FUNCTION_BLOCK Jack_Sledge_Place (* Composite Function Block Type *)
  (* Standard: 61499-2 *)
  (* Version 0.0, 4/24/2020, prana, nxtControl GmbH, template *)
  PACKAGE Main;
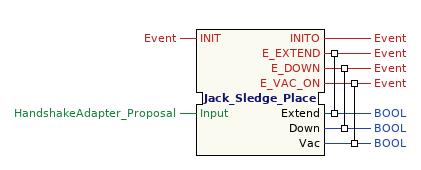
  EVENT_INPUT
    INIT; (* Initialization Request *)
  END_EVENT
  EVENT_OUTPUT
    INITO; (* Initialization Confirm *)
    E_EXTEND WITH Extend;
    E_DOWN WITH Down;
    E_VAC_ON WITH Vac;
  END_EVENT
  VAR_OUTPUT
    Extend : BOOL;
    Down : BOOL;
    Vac : BOOL;
  END_VAR
  SOCKETS
    Input : HandshakeAdapter_Proposal;
  END_SOCKETS
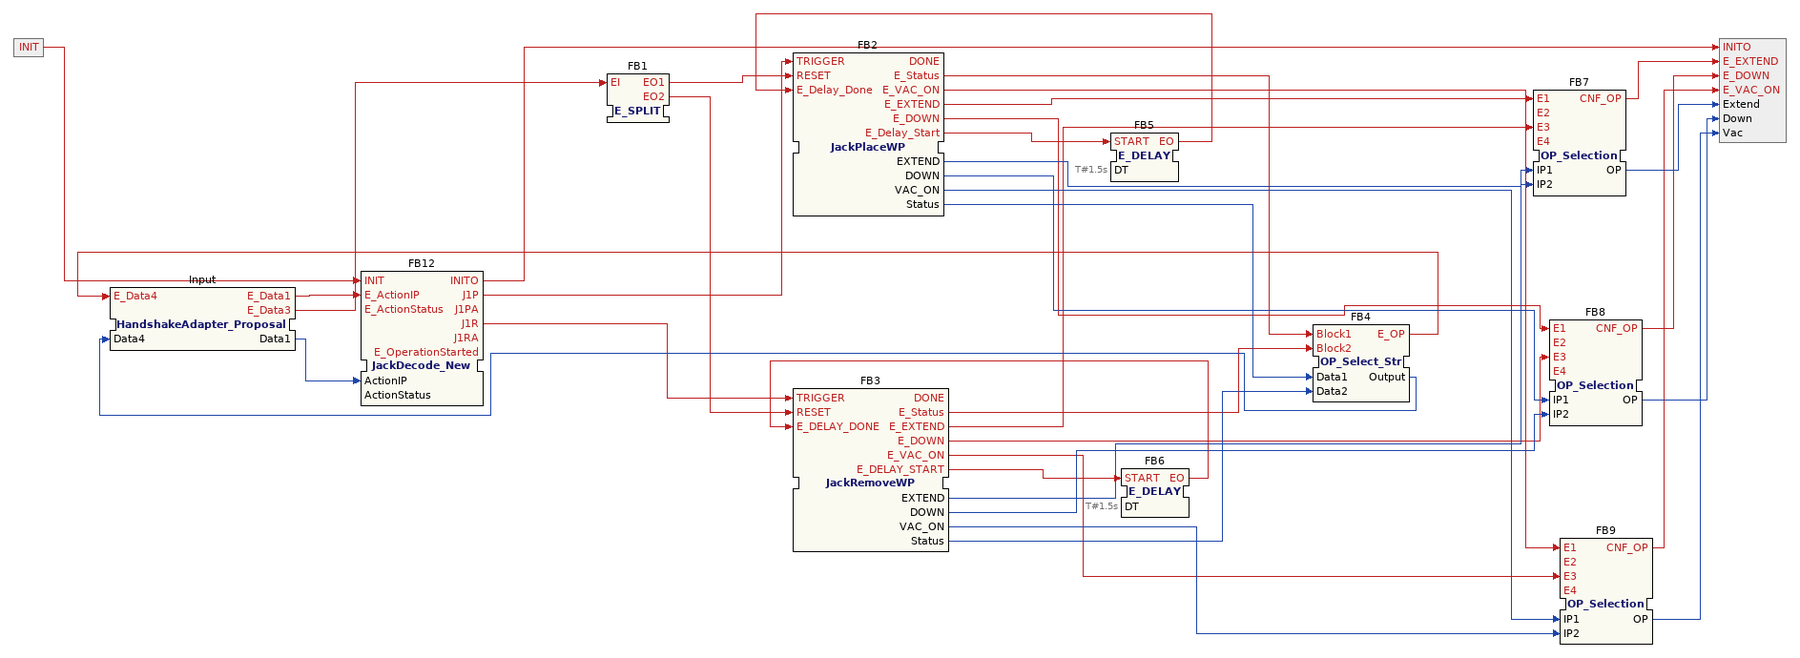
  FBS
    FB1 : E_SPLIT;
    FB12 : JackDecode_New;
    FB2 : JackPlaceWP;
    FB3 : JackRemoveWP;
    FB4 : OP_Select_Str;
    FB5 : E_DELAY(DT := T#1.5s);
    FB6 : E_DELAY(DT := T#1.5s);
    FB7 : OP_Selection;
    FB8 : OP_Selection;
    FB9 : OP_Selection;
  END_FBS
  EVENT_CONNECTIONS
    Input.E_Data1 TO FB12.E_ActionIP;
    INIT TO FB12.INIT;
    FB1.EO1 TO FB2.RESET;
    FB1.EO2 TO FB3.RESET;
    FB12.INITO TO INITO;
    FB12.J1P TO FB2.TRIGGER;
    FB12.J1R TO FB3.TRIGGER;
    FB2.E_Status TO FB4.Block1;
    FB3.E_Status TO FB4.Block2;
    FB4.E_OP TO Input.E_Data4;
    FB5.EO TO FB2.E_Delay_Done;
    FB2.E_Delay_Start TO FB5.START;
    FB3.E_DELAY_START TO FB6.START;
    FB6.EO TO FB3.E_DELAY_DONE;
    FB2.E_EXTEND TO FB7.E1;
    FB3.E_EXTEND TO FB7.E3;
    FB2.E_DOWN TO FB8.E1;
    FB3.E_DOWN TO FB8.E3;
    FB3.E_VAC_ON TO FB9.E3;
    FB2.E_VAC_ON TO FB9.E1;
    FB8.CNF_OP TO E_DOWN;
    FB9.CNF_OP TO E_VAC_ON;
    FB7.CNF_OP TO E_EXTEND;
    Input.E_Data3 TO FB1.EI;
  END_CONNECTIONS
  DATA_CONNECTIONS
    Input.Data1 TO FB12.ActionIP;
    FB2.Status TO FB4.Data1;
    FB3.Status TO FB4.Data2;
    FB4.Output TO Input.Data4;
    FB7.OP TO Extend;
    FB8.OP TO Down;
    FB9.OP TO Vac;
    FB2.EXTEND TO FB7.IP1;
    FB3.EXTEND TO FB7.IP2;
    FB2.DOWN TO FB8.IP1;
    FB3.DOWN TO FB8.IP2;
    FB3.VAC_ON TO FB9.IP2;
    FB2.VAC_ON TO FB9.IP1;
  END_CONNECTIONS
END_FUNCTION_BLOCK
